(* CODESYS project PLC 1 Simulatie Structured Tekst 2V0 - Leeg.project
   Company: Avans
   Description: Simulatie voor opstelling Sorteer Station.
   Title: Simulatie Sorteer Station
   Author: Rene Potters/Gerard Harkema
   Version: 0.1.0

Project tree, tasks and I/O mapping:
  Device : CODESYS Control Win V3, 3S - Smart Software Solutions GmbH, version 3.5.13.20
    application SorteerStationSimulatie
      libraries: Standard, * (System); Util, * (System); VisuDialogs, 3.5.12.0 (System)
      task MainTask (cyclic, interval t#20ms, priority 1) calls Main
      task Simulatie (cyclic, interval t#20ms, priority 1) calls MagazijnSim, OverzetterSim, SorterenSim
  Device_1 : EHV-CPU1025, Hitachi-IES, order no. EHV-CPU1025, version 3.5.4.11
      settings: IP Address = '192.168.1.31'
    application SorteerStationRealWorld
      libraries: Standard, * (System); Util, * (System); VisuDialogs, 3.5.12.0 (System)
      task MainTask (cyclic, interval t#20ms, priority 1) calls Main
    Basic : Basic, Hitachi-IES, version 3.4.4.0
      <Empty>
      <Empty>
      <Empty>
      <Empty>
      <Empty>
      <Empty>
      <Empty>
      <Empty>
      <Empty>
      <Empty>
      <Empty>
  Simulatie/
    program MagazijnSim [ST]
    program SorterenSim [ST]
    global variables SIM
    program OverzetterSim [ST]
    data type OverzetterDUT
    data type SorterenDUT
    data type MagazijnDUT
    function block SorterenGootSim [ST]
  text list GlobalTextList
  Programma Structured Text/
    program Main [ST]
  global variables GVL
  Visualisaties/
    visualisation SorteerStationHMI
    visualisation BekerMagazijnHMI
    visualisation OverzetterHMI
    visualisation SorterenHMI
*)

// Simulatie/OverzetterDUT
{attribute 'qualified_only'}
{attribute 'strict'}
TYPE OverzetterDUT :
(
	INHETMIDDEN, NAARRECHTS, ISRECHTS, NAARLINKS, ISLINKS, GEVALLEN
);
END_TYPE

// Simulatie/SorterenDUT
{attribute 'qualified_only'}
{attribute 'strict'}
TYPE SorterenDUT :
(
	VOLGENDEBLOK, OPDEBAND, VOORSTOPPER, NAARGOOT1, INGOOT1, NAARGOOT2, INGOOT2, NAARGOOT3, INGOOT3, GEREED, VOL
);
END_TYPE

// Simulatie/MagazijnDUT
{attribute 'qualified_only'}
{attribute 'strict'}
TYPE MagazijnDUT :
(
	INGETROKKEN, INTREKKEN, UITGESTOTEN, UITSTOTEN, LEEG
);
END_TYPE

// Simulatie/SIM
{attribute 'qualified_only'}
VAR_GLOBAL
	// Rotatie van de overzetter
	Vx_OvzRotate: INT := 0;
	// Visualisatie invisible blok
	Vx_OvzBlokLinks: BOOL := FALSE;
	// Visualisatie invisible blok
	Vx_OvzBlokOverzetter: BOOL := FALSE;
	// Visualisatie invisible blok
	Vx_OvzBlokRechts: BOOL := FALSE;
	// Visualisatie invisible blok
	Vx_OvzBlokGevallen: BOOL := FALSE;	
	// Magazijn opnieuw vullen (simulatie)
	Ix_MagazijnVullen 	: BOOL;
	// Goten legen (symulatie)
	Ix_GotenLegen	  	: BOOL;
	
	
	
	
	
	
	
	
	
	
	
	
	
	
	
	
	
	
	
	
	
	
	
	
	
	
	
	
	
	
	
	
	
	
	
	
	
	
	
	
	
	
	
	
	
	
	
	
	// Simulatie visualisatie 
	Vw_Rotate45: INT := 45;
	// Visualisatie X positie van de uitstoter
	Vw_MagUitstoterBekerX: INT := 30;
	// Visualisatie invisible blok uitgestoten
	Vx_MagBlokUit: BOOL := TRUE;
	// Visualisatie invisible blok 1
	Vx_MagBlok1: BOOL := TRUE;
	// Visualisatie invisible blok 2
	Vx_MagBlok2: BOOL := TRUE;
	// Visualisatie invisible blok 3
	Vx_MagBlok3: BOOL := TRUE;
	// Visualisatie invisible blok 4
	Vx_MagBlok4: BOOL := TRUE;
	// Visualisatie invisible blokken
	Vx_MagBlok: ARRAY[1..8] OF BOOL;
	// Aantal blokken in het magazijn
	Vw_MagBlokAantal: INT := 4;
	// Simulatie onthoudt dat een blok maar 1x wordt uitgestoten
	Vw_MagBlok1X: INT := 0;
	// Ligt er een blok op band
	Vw_SorBlokBand: BOOL := FALSE;
	// Rotatie van de stopper
	Vw_SorStopperRotate: INT := 0;
	// Rotatie van de stopper goot 1
	Vw_SorGoot1Rotate: INT := 0;
	// Rotatie van de stopper goot 2
	Vw_SorGoot2Rotate: INT := 0;
	// Kleur van de blok op betreffende positie
	Vw_SorKleurBand: DWORD := 0;
	// Bewegen van de blok over de band
	Vi_SorBlokBandX: INT := 0;
	// Bewegen van de blok over de band
	Vi_SorBlokBandY: INT := 0;
	// Simulatie error. Inverse logica.
	Vx_MagLuchtDrukError: BOOL := TRUE;
	// Simulatie error. Inverse logica.
	Vx_MagIsInError: BOOL := TRUE;
	// Simulatie error. Inverse logica.
	Vx_MagIsUitError: BOOL := TRUE;
	// Simulatie error. Inverse logica.
	Vx_OvzLuchtDrukError: BOOL := TRUE;
	// Simulatie error. Inverse logica.
	Vx_OvzIsLinksError: BOOL := TRUE;
	// Simulatie error. Inverse logica.
	Vx_OvzIsRechtsError: BOOL := TRUE;
	// Simulatie error. Inverse logica.
	Vx_OvzVacuumError: BOOL := TRUE;
	// Simulatie error. Inverse logica.
	Vx_SorMotorAfvoerError: BOOL := TRUE;
	// Simulatie error. Inverse logica.
	Vx_SorGoot1InError: BOOL := TRUE;
	// Simulatie error. Inverse logica.
	Vx_SorGoot1UitError: BOOL := TRUE;
	// Simulatie error. Inverse logica.
	Vx_SorInGootError: BOOL := TRUE;
	// Ligt er een blok op de betreffende positie
	Vx_SorBlokGoot: ARRAY [1..3,1..6] OF BOOL;
	// Kleur van de blok op betreffende positie
	Vw_SorKleurGoot: ARRAY [1..3,1..6] OF DWORD;
END_VAR

// GVL
VAR_GLOBAL
	// Indrukken resetknop 
	Ix_Resetknop: BOOL;
	// Keuzeknop staat op hand
	Ix_Hand: BOOL;
	// Keuzeknop staat op auto
	Ix_Auto: BOOL;
	// Indrukken noodstop
	Ix_Noodstop: BOOL;
	// Bekers magazijn zijn op
	Ix_MagazijnLeeg: BOOL;
	// Beker is uit dekselmagazijn gestoten
	Ix_UitstoterBekerIn: BOOL;
	// Uitstoter Beker haalt nieuwe beker op
	Ix_UitstoterBekerUit: BOOL;
	// Indrukken startknop
	Ix_Stopknop: BOOL := TRUE;
	// Indrukken stopknop
	Ix_Startknop: BOOL;	
	//Perslucht is aanwezig
	Ix_PersluchtAanwezig :BOOL;
	//Werkstuk door overzetter opgepakt
	Ix_VacuumAanwezig :BOOL;
	//Overzetter haalt beker op(linker pos.)
	Ix_OverzetterIsLinks :BOOL;
	//Overzetter plaatst beker op sorteerpositie
	Ix_OverzetterIsRechts :BOOL;
	//Beker aanwezig op detectiepositie
	Ix_BekerAanwezig :BOOL;
	//Beker is van aluminium
	Ix_BekerMetaal :BOOL;
	//Beker reflecteert en is dus niet zwart
	Ix_BekerReflecteerd :BOOL;
	//Product is naar een van de goten gegaan
	Ix_BekerInGoot :BOOL;
	//Pusher uitvoergoot 1 is in
	Ix_UitvoerGoot1IsIn :BOOL;
	//Pusher uitvoergoot 2 is in
	Ix_UitvoerGoot2IsIn :BOOL;
	//Beker afvoeren is bezig
	Ix_StationAfvoerVrij :BOOL;
	//Pusher uitvoergoot 1 is uit
	Ix_UitvoerGoot1IsUit :BOOL;
	//Pusher uitvoergoot 2 is uit
	Ix_UitvoerGoot2IsUit :BOOL;
	// Beker uit magazijn stoten
	Qx_BekerUitstoten: BOOL;	
	//Beker oppakken
	Qx_VacuumAan :BOOL;
	//Beker loslaten
	Qx_BekerLossen :BOOL;
	//Overzetter naar bekermagazijn
	Qx_OverzetterLinks :BOOL;
	//Overzetter naar sorteerpositie
	Qx_OverzetterRechts :BOOL;
	//Transportband aan
	Qx_MotorAfvoerAan :BOOL;
	//Pusher goot 1 uit
	Qx_UitvoerGoot1Uit :BOOL;
	//Pusher goot 2 uit
	Qx_UitvoerGoot2Uit :BOOL;
	//Beker stoppen op band voor detectie
	Qx_StopperUit :BOOL;
	//Uitsorteren is bezet
	Qx_StationBezet :BOOL;
	// Visualisatie invisible Gele vlak
	Qx_GeleLamp: BOOL;
	// Visualisatie invisible groene vlak
	Qx_GroeneLamp: BOOL;
	// Visualisatie invisible rode vlak
	Qx_RodeLamp: BOOL;
END_VAR

// Programma Structured Text/Main
PROGRAM Main
VAR
END_VAR

END_PROGRAM

// Simulatie/MagazijnSim
PROGRAM MagazijnSim
VAR
	// Timer om uitstoten en intrekken te vertragen
	Fb_Pulse: BLINK;
	// Timer om intrekken te vertragen
	Fb_Trigger: F_TRIG;
	// Eerste keer om visualisatie te updaten
	Mx_FirstTime: BOOL := TRUE;
	// Afhandeling van het magazijn
	Me_MagState: MAGAZIJNDUT := MAGAZIJNDUT.INGETROKKEN;
END_VAR

//
// Common stuff.
//

IF (Mx_FirstTime) THEN
	SIM.Vw_MagBlokAantal := 8;
	SIM.Vx_MagBlokUit:= FALSE;
	
	Mx_FirstTime := FALSE;
END_IF

					
//
// Handle all pulse and trigger events.
//
Fb_Pulse(ENABLE:=TRUE,TIMELOW:=T#200MS, TIMEHIGH:=T#200MS);
Fb_Trigger(CLK:=Fb_Pulse.OUT);


//
// Only if no emergency active, start handling the simulation.
//
IF (SIM.Ix_MagazijnVullen) THEN
	Mx_FirstTime := TRUE;
	SIM.Ix_MagazijnVullen := FALSE;
	RETURN;
END_IF
	
//
// The pulse determines the speed of the cilinder to move in
// ore move out. The cilinder is only moved if the airpressure 
// is available.
//
IF (Fb_Trigger.Q AND SIM.Vx_MagLuchtDrukError) THEN
		
			
	CASE Me_MagState OF
		MAGAZIJNDUT.INGETROKKEN:
			IF (SIM.Vx_MagBlokUit) THEN
				SIM.Vw_MagBlokAantal := SIM.Vw_MagBlokAantal - 1;
			END_IF
		
			SIM.Vw_MagUitstoterBekerX := 1;
			SIM.Vw_MagBlok1X    	  := SIM.Vw_MagUitstoterBekerX;
			SIM.Vx_MagBlokUit         := FALSE;
	
			IF (Qx_BekerUitstoten) THEN
				Me_MagState := MAGAZIJNDUT.UITSTOTEN;
			END_IF

		MAGAZIJNDUT.INTREKKEN:
			SIM.Vw_MagUitstoterBekerX := SIM.Vw_MagUitstoterBekerX - 30;
			
			IF (SIM.Vw_MagUitstoterBekerX < 0) THEN 
				SIM.Vw_MagUitstoterBekerX := 0; 
			END_IF		
			
			IF (SIM.Vw_MagUitstoterBekerX = 0) THEN
				Me_MagState := MAGAZIJNDUT.INGETROKKEN;				
			END_IF		

			IF (Qx_BekerUitstoten) THEN
				Me_MagState := MAGAZIJNDUT.UITSTOTEN;
			END_IF	
	
		MAGAZIJNDUT.UITGESTOTEN:
			SIM.Vx_MagBlokUit         := SIM.Vx_MagBlok1;
						
			IF (NOT Qx_BekerUitstoten) THEN
				Me_MagState := MAGAZIJNDUT.INTREKKEN;
			END_IF	
		
		MAGAZIJNDUT.UITSTOTEN:
			SIM.Vw_MagUitstoterBekerX := SIM.Vw_MagUitstoterBekerX + 30;
			SIM.Vw_MagBlok1X    	  := SIM.Vw_MagUitstoterBekerX;			
		
			IF (SIM.Vw_MagUitstoterBekerX > 70) THEN
				Me_MagState := MAGAZIJNDUT.UITGESTOTEN;				
			END_IF		

			IF (NOT Qx_BekerUitstoten) THEN
				Me_MagState := MAGAZIJNDUT.INTREKKEN;
			END_IF	
		
	END_CASE

	GVL.Ix_UitstoterBekerIn  := (Me_MagState = MAGAZIJNDUT.INGETROKKEN) AND SIM.Vx_MagIsInError;
	GVL.Ix_UitstoterBekerUit := (Me_MagState = MAGAZIJNDUT.UITGESTOTEN) AND SIM.Vx_MagIsUitError;	
	GVL.Ix_MagazijnLeeg 	 := (SIM.Vw_MagBlokAantal <= 0) AND (Ix_UitstoterBekerIn);	
	
	SIM.Vx_MagBlok[8] := (SIM.Vw_MagBlokAantal >= 8);
	SIM.Vx_MagBlok[7] := (SIM.Vw_MagBlokAantal >= 7);
	SIM.Vx_MagBlok[6] := (SIM.Vw_MagBlokAantal >= 6);
	SIM.Vx_MagBlok[5] := (SIM.Vw_MagBlokAantal >= 5);		
	SIM.Vx_MagBlok[4] := (SIM.Vw_MagBlokAantal >= 4);
	SIM.Vx_MagBlok[3] := (SIM.Vw_MagBlokAantal >= 3);
	SIM.Vx_MagBlok[2] := (SIM.Vw_MagBlokAantal >= 2);
	SIM.Vx_MagBlok[1] := (SIM.Vw_MagBlokAantal >= 1);	
	
END_IF

END_PROGRAM

// Simulatie/OverzetterSim
PROGRAM OverzetterSim
VAR
	// Timer om overzetten te vertragen
	Fb_Pulse: BLINK;
	// Timer om overzetten te vertragen
	Fb_Trigger: F_TRIG;
	// Eerste keer om visualisatie te updaten
	Mx_FirstTime: BOOL := TRUE;
	// Afhandeling van de overzetter
	Me_OvzState: OverzetterDUT := OVERZETTERDUT.INHETMIDDEN;	
	// Afhandeling van het blokje
	Me_BlokState: OverzetterDUT := OVERZETTERDUT.INHETMIDDEN;	
	// Duurt even voor het vacuum aanwezig is
	Mi_VacuumCntr: INT := 0;	
END_VAR
VAR CONSTANT


	// Inverse logica
	INVISABLE: BOOL := TRUE;
	// Inverse logica
	VISABLE: BOOL := FALSE;

END_VAR

// Initialisatie.

IF (Mx_FirstTime) THEN
	Me_OvzState := OVERZETTERDUT.INHETMIDDEN;
	Me_BlokState := OVERZETTERDUT.ISLINKS;
	
	Mi_VacuumCntr := 0;
	SIM.Vx_OvzRotate := 0;
	Mx_FirstTime := FALSE;
END_IF

//
// Afhandelen van de pulse events. Hierdoor loopt de simulatie los van de 
// TASK tijd.
//
Fb_Pulse(ENABLE:=TRUE,TIMELOW:=T#100MS, TIMEHIGH:=T#100MS);
Fb_Trigger(CLK:=Fb_Pulse.OUT);


//
// Only if no emergency active, start handling the simulation.
//
IF (GVL.Ix_Noodstop) THEN
	Mx_FirstTime := TRUE;	
	RETURN;
END_IF
	
//
// The pulse determines the speed of the cilinder to move in
// ore move out. The cilinder is only moved if the airpressure 
// is available.
//
IF (Fb_Trigger.Q AND SIM.Vx_OvzLuchtDrukError) THEN
	
	//
	// De status van de arm wordt los afgehandeld van het blokje. De beweging
	// van de arm staat hier namelijk helemaal los van.
	//
	
	CASE Me_OvzState OF
		
		OVERZETTERDUT.INHETMIDDEN:
			// 
			// De arm is in beweging naar links of naar rechts.
			// Indien de arm in de uiterste positie is wordt er van 
			// state gewisseld. Aangezien de arm in beweging is staan
			// de eindschakelaars uit.
			//
			
			IF (GVL.Qx_OverzetterLinks) THEN
				IF (SIM.Vx_OvzRotate > -90) THEN
					GVL.Ix_OverzetterIsLinks := FALSE;	
					GVL.Ix_OverzetterIsRechts := FALSE;			
					SIM.Vx_OvzRotate := SIM.Vx_OvzRotate - 10;
				ELSE
					Me_OvzState := OVERZETTERDUT.ISLINKS;			
				END_IF	
				
			END_IF
				 
			IF (GVL.Qx_OverzetterRechts) THEN
				IF (SIM.Vx_OvzRotate < 90) THEN
					GVL.Ix_OverzetterIsLinks := FALSE;	
					GVL.Ix_OverzetterIsRechts := FALSE;				
					SIM.Vx_OvzRotate := SIM.Vx_OvzRotate + 10;
				ELSE
					Me_OvzState := OVERZETTERDUT.ISRECHTS;				
				END_IF			
			END_IF
				
		OVERZETTERDUT.ISLINKS:
		    //
			// Arm staat in een uiterste stand. Eindschakelaar is ingeschakeld.
			// Zodra de arm weer wordt bewogen verandert de state.
			//
			
			GVL.Ix_OverzetterIsLinks := TRUE AND SIM.Vx_OvzIsLinksError;	

			IF (GVL.Qx_OverzetterRechts AND NOT GVL.Qx_OverzetterLinks) THEN
				GVL.Ix_OverzetterIsLinks := FALSE;				
				Me_OvzState := OVERZETTERDUT.INHETMIDDEN;		
			END_IF
			
		OVERZETTERDUT.ISRECHTS:
		    //
			// Arm staat in een uiterste stand. Eindschakelaar is ingeschakeld.
			// Zodra de arm weer wordt bewogen verandert de state.
			//
		
			GVL.Ix_OverzetterIsRechts := TRUE AND SIM.Vx_OvzIsRechtsError;	

			IF (GVL.Qx_OverzetterLinks AND NOT GVL.Qx_OverzetterRechts) THEN
				GVL.Ix_OverzetterIsRechts := FALSE;				
				Me_OvzState := OVERZETTERDUT.INHETMIDDEN;		
			END_IF			
			
		END_CASE

	END_IF	

	//
	// De status van het blokje hangt af van een aantal stuursignalen zoals waar
	// de arm zich bevindt, of er vacuum is en of er een beker lossen wordt gegeven.
	//
	
	CASE Me_BlokState OF
		OVERZETTERDUT.ISLINKS:
			//
			// Als de arm links is moet er eerste een vacuum opgebouwd worden alvorens het blokje 
			// opgepakt kan worden. Daarna verandert de state. 
			//
			
			SIM.Vx_OvzBlokGevallen 	 := INVISABLE;
			SIM.Vx_OvzBlokLinks 	 := VISABLE;
			SIM.Vx_OvzBlokOverzetter := INVISABLE;
			SIM.Vx_OvzBlokRechts 	 := INVISABLE;
			
			IF (GVL.Qx_VacuumAan AND SIM.Vx_OvzVacuumError AND GVL.Ix_OverzetterIsLinks) AND (NOT GVL.Qx_BekerLossen) THEN
				Mi_VacuumCntr := Mi_VacuumCntr + 1;
			END_IF
			
			IF (NOT GVL.Qx_VacuumAan AND SIM.Vx_OvzVacuumError) THEN
				Mi_VacuumCntr := 0;
			END_IF

			GVL.Ix_VacuumAanwezig := (Mi_VacuumCntr > 50);
	
			IF  ( GVL.Ix_VacuumAanwezig AND (Me_OvzState = OVERZETTERDUT.INHETMIDDEN)) THEN
				Me_BlokState := OVERZETTERDUT.INHETMIDDEN;
			END_IF
			
		OVERZETTERDUT.INHETMIDDEN:
			//
			// Het blokje is in beweging zolang er vacuum is. Als er geen vacuum meer is
			// valt het blokje... Indien de arm helemaal rechts is kan het blokje gelost 
			// worden. Dit moet met een Bekerlossen ondanks het feit dat er
			// geen vacuum meer is....
			//
			
			SIM.Vx_OvzBlokGevallen 	 := INVISABLE;
			SIM.Vx_OvzBlokLinks 	 := INVISABLE;
			SIM.Vx_OvzBlokOverzetter := VISABLE;
			SIM.Vx_OvzBlokRechts 	 := INVISABLE;

		 	IF (GVL.Ix_OverzetterIsRechts) AND (NOT GVL.Qx_VacuumAan) AND (GVL.Qx_BekerLossen) THEN
				GVL.Ix_VacuumAanwezig := FALSE;
				Me_BlokState := OVERZETTERDUT.ISRECHTS;		
				RETURN;		
			END_IF
			
			IF (NOT GVL.Ix_OverzetterIsRechts) AND (NOT GVL.Ix_OverzetterIsLinks) AND(NOT GVL.Qx_VacuumAan) THEN
				GVL.Ix_VacuumAanwezig := FALSE;
				Me_BlokState := OVERZETTERDUT.GEVALLEN;				
			END_IF

		OVERZETTERDUT.ISRECHTS:	
		    // 
			// Blokje is gelost. Nu is het wachten tot de overzetter terug naar links wordt gestuurd. Daarna verdwijnt
			// het blokje automatisch.
			//
			
			SIM.Vx_OvzBlokGevallen 	 := INVISABLE;
			SIM.Vx_OvzBlokLinks 	 := INVISABLE;
			SIM.Vx_OvzBlokOverzetter := INVISABLE;
			SIM.Vx_OvzBlokRechts 	 := VISABLE;
			
			IF (NOT GVL.Ix_OverzetterIsRechts) THEN
				Me_BlokState := OVERZETTERDUT.ISLINKS;					
			END_IF

		OVERZETTERDUT.GEVALLEN:
			//
			// Blokje is gevallen..... Situatie herstelt zich zodra de arm helemaal links staat.
			//
				
			SIM.Vx_OvzBlokGevallen 	 := VISABLE;
			SIM.Vx_OvzBlokLinks 	 := INVISABLE;
			SIM.Vx_OvzBlokOverzetter := INVISABLE;
			SIM.Vx_OvzBlokRechts 	 := INVISABLE;
			
			IF (GVL.Ix_OverzetterIsLinks) THEN
				Me_BlokState := OVERZETTERDUT.ISLINKS;					
			END_IF				
	END_CASE

END_PROGRAM

// Simulatie/SorterenSim
PROGRAM SorterenSim
VAR
	// Timer om sorteren te vertragen
	Fb_Pulse: BLINK;
	// Timer om sorteren te vertragen
	Fb_Trigger: F_TRIG;
	// Eerste keer om visualisatie te updaten
	Mx_FirstTime: BOOL := TRUE;
	// Afhandeling van de overzetter
	Me_SorState: SORTERENDUT := SORTERENDUT.OPDEBAND;
	// Index voor posities
	Mi_PositieIndx: INT := 1;
	// Index voor goten.
	Mi_GootIndx: INT := 1;
	// Afhandeling blokjes in goot1.
	Mb_Goot1: SorterenGootSim;
	// Afhandeling blokjes in goot2.
	Mb_Goot2: SorterenGootSim;
	// Afhandeling blokjes in goot3.
	Mb_Goot3: SorterenGootSim;
	Mx_Geplaatst: BOOL := FALSE;
	// Random nummer om kleur te bepalen
	Mi_Random: UDINT := 1;	
END_VAR
VAR CONSTANT
	// Inverse logica
	INVISABLE: BOOL := TRUE;
	// Inverse logica
	VISABLE: BOOL := FALSE;
	// Kleur rood
	RED: DWORD := 16#00FF0000;
	// Kleur wit
	WHITE: DWORD := 16#00FFFFFF;
	// Stapgrootte voor bewegingen
	STEP: INT := 4;
	// Kleur zwart
	BLACK: DWORD := 16#00000000;
	// Kleur geel
	YELLOW: DWORD := 16#00FFFF00;
	// Goot 1
	GOOT1: INT := 1;
	// Goot 2
	GOOT2: INT := 2;
	// Goot 3
	GOOT3: INT := 3;
END_VAR

// Initialisatie.

IF (Mx_FirstTime) THEN
	Me_SorState := SORTERENDUT.VOLGENDEBLOK;

	SIM.Vw_SorBlokBand  := VISABLE;
	SIM.Vw_SorKleurBand := YELLOW;
	SIM.Vi_SorBlokBandX := 0;
	SIM.Vi_SorBlokBandY := 0;
	
	FOR Mi_GootIndx := 1 TO 3 DO 
		FOR Mi_PositieIndx := 1 TO 3 DO
			SIM.Vx_SorBlokGoot[Mi_GootIndx, Mi_PositieIndx ]  := INVISABLE;
			SIM.Vw_SorKleurGoot[Mi_GootIndx, Mi_PositieIndx ] := WHITE;			
		END_FOR
	END_FOR
 
	Mx_FirstTime := FALSE;
END_IF

//
// Afhandelen van de pulse events. Hierdoor loopt de simulatie los van de 
// TASK tijd.
//
Fb_Pulse(ENABLE:=TRUE,TIMELOW:=T#50MS, TIMEHIGH:=T#50MS);
Fb_Trigger(CLK:=Fb_Pulse.OUT);


//
// Only if no emergency active, start handling the simulation.
//
IF (SIM.Ix_GotenLegen) THEN
	Mx_FirstTime := TRUE;
	SIM.Ix_GotenLegen := FALSE;
	RETURN;
END_IF


// The pulse determines the speed of the cilinder to move in
// ore move out. The cilinder is only moved if the airpressure 
// is available.
//
IF (Fb_Trigger.Q) THEN
	IF (GVL.Qx_StopperUit) THEN
		SIM.Vw_SorStopperRotate := 90;
	ELSE
		SIM.Vw_SorStopperRotate := 0;		
	END_IF
	
	IF (GVL.Qx_UitvoerGoot1Uit) THEN
		SIM.Vw_SorGoot1Rotate := 45;
	ELSE
		SIM.Vw_SorGoot1Rotate := 0;		
	END_IF	

	GVL.Ix_UitvoerGoot1IsUit := (SIM.Vw_SorGoot1Rotate > 0) AND (SIM.Vx_SorGoot1UitError);
    GVL.Ix_UitvoerGoot1IsIn  := (SIM.Vw_SorGoot1Rotate = 0) AND (SIM.Vx_SorGoot1InError);	
	
	IF (GVL.Qx_UitvoerGoot2Uit) THEN
		SIM.Vw_SorGoot2Rotate := 45;
	ELSE
		SIM.Vw_SorGoot2Rotate := 0;		
	END_IF	

	GVL.Ix_UitvoerGoot2IsUit := (SIM.Vw_SorGoot2Rotate > 0);
    GVL.Ix_UitvoerGoot2IsIn  := (SIM.Vw_SorGoot2Rotate = 0);	
	
	GVL.Ix_BekerInGoot := SIM.Vx_SorInGootError AND NOT ((SIM.Vx_SorBlokGoot[1,1] = VISABLE) OR (SIM.Vx_SorBlokGoot[2,1] = VISABLE) OR (SIM.Vx_SorBlokGoot[3,1] = VISABLE) OR ((SIM.Vi_SorBlokBandY > 30) AND (SIM.Vi_SorBlokBandY < 40)));


				
	CASE Me_SorState OF
		SORTERENDUT.VOLGENDEBLOK:
			//
			// Zet alles klaar voor een volgende blokje.
			//

			Mi_Random := DINT_TO_UDINT(TIME_TO_DINT(TIME()));
			Mi_Random := SHR((Mi_Random AND 16#000000F00), 8); 
   
			IF (Mi_Random < 5) THEN
				SIM.Vw_SorKleurBand := RED;
			ELSE IF (Mi_Random < 10) THEN
					SIM.Vw_SorKleurBand := BLACK;
				ELSE 
					SIM.Vw_SorKleurBand := YELLOW;
				END_IF
			END_IF
			
			SIM.Vw_SorBlokBand := VISABLE;
			SIM.Vi_SorBlokBandX := 0;
			SIM.Vi_SorBlokBandY := 0;
	
			Me_SorState := SORTERENDUT.OPDEBAND;
		
		SORTERENDUT.OPDEBAND:
		
			//
			// Blokje ligt op de band. Verplaats tot voor de stopper.
			//
			
			IF ((GVL.Qx_MotorAfvoerAan) AND (SIM.Vx_SorMotorAfvoerError)) THEN
				SIM.Vi_SorBlokBandX := SIM.Vi_SorBlokBandX + STEP;
			END_IF
			
			GVL.Ix_StationAfvoerVrij := (SIM.Vi_SorBlokBandX < 20);
			
			IF (SIM.Vi_SorBlokBandX > 50) THEN
				Me_SorState := SORTERENDUT.VOORSTOPPER;
			END_IF
			
		SORTERENDUT.VOORSTOPPER: 
		
			//
			// Indien de stopper uit is, dan stopt het blokje en worden
			// de kleur sensoren geactiveerd. Anders loopt het blokje gewoon door
			// naar goot 1.
			//
			
			IF ((NOT GVL.Qx_StopperUit) AND (GVL.Qx_MotorAfvoerAan) AND (SIM.Vx_SorMotorAfvoerError)) THEN
				SIM.Vi_SorBlokBandX := SIM.Vi_SorBlokBandX + STEP;	
			END_IF

			IF (GVL.Qx_StopperUit) THEN
				GVL.Ix_BekerAanwezig := TRUE;
				GVL.Ix_BekerMetaal       := (SIM.Vw_SorKleurBand = YELLOW);
				GVL.Ix_BekerReflecteerd  := (SIM.Vw_SorKleurBand = YELLOW) OR (SIM.Vw_SorKleurBand = RED);
			END_IF
			
			
			IF (SIM.Vi_SorBlokBandX > 60) THEN
				Me_SorState := SORTERENDUT.NAARGOOT1;
			END_IF		
		
		
		SORTERENDUT.NAARGOOT1:
			//
			// Voor goot 1 wordt bepaald of de stopper uit staat en het blokje dus in de goot
			// gaat. Anders loopt het blokje door naar goot 2.
			//

			GVL.Ix_BekerAanwezig := FALSE;
			
			IF ((GVL.Qx_MotorAfvoerAan) AND (SIM.Vx_SorMotorAfvoerError)) THEN
				SIM.Vi_SorBlokBandX := SIM.Vi_SorBlokBandX + STEP;
			END_IF
			
			IF ((SIM.Vi_SorBlokBandX > 130) AND (GVL.Qx_MotorAfvoerAan) AND (SIM.Vx_SorMotorAfvoerError) AND (GVL.Qx_UitvoerGoot1Uit)) THEN
				Me_SorState := SORTERENDUT.INGOOT1;
			END_IF		
	
			IF ((SIM.Vi_SorBlokBandX > 130) AND (GVL.Qx_MotorAfvoerAan) AND (SIM.Vx_SorMotorAfvoerError) AND (NOT GVL.Qx_UitvoerGoot1Uit)) THEN
				Me_SorState := SORTERENDUT.NAARGOOT2;
			END_IF	
	 
		SORTERENDUT.INGOOT1:
			//
			// Blokje valt in goot 1. Hier kunnen 3 blokjes liggen. Het  blokje van de band beweegt de goot 
			// in en aan de hand van welke blokjes er al liggen wordt het eerst volgende blokje bepaald.
			// Dit blokje wordt vervolgens getoond. Daarna is het sorteren gereed. Let op dat de goot vol
			// melding even wordt getriggered als het blokje door de sensor valt.
			//
			
			IF (SIM.Vi_SorBlokBandX < 170) THEN
				SIM.Vi_SorBlokBandX := SIM.Vi_SorBlokBandX + 2*STEP;
			END_IF
			
			SIM.Vi_SorBlokBandY := SIM.Vi_SorBlokBandY + STEP;

			
			Mb_Goot1(Px_YPos:=SIM.Vi_SorBlokBandY, Px_Goot:=GOOT1);
		
			IF (Mb_Goot1.Px_Geplaatst) THEN
				Me_SorState := SORTERENDUT.GEREED;
			END_IF
			
			IF (SIM.Vx_SorBlokGoot[GOOT1, 1] = VISABLE) THEN
				Me_SorState := SORTERENDUT.VOL;
			END_IF
			
		SORTERENDUT.NAARGOOT2: 
			//
			// Voor goot 2 wordt bepaald of de stopper uit staat en het blokje dus in de goot
			// gaat. Anders loopt het blokje door naar goot 3.
			//
		
			IF ((GVL.Qx_MotorAfvoerAan) AND (SIM.Vx_SorMotorAfvoerError)) THEN
				SIM.Vi_SorBlokBandX := SIM.Vi_SorBlokBandX + STEP;
			END_IF
			
			IF ((SIM.Vi_SorBlokBandX > 230) AND (GVL.Qx_MotorAfvoerAan) AND (SIM.Vx_SorMotorAfvoerError) AND (GVL.Qx_UitvoerGoot2Uit)) THEN
				Me_SorState := SORTERENDUT.INGOOT2;
			END_IF		
	
			IF ((SIM.Vi_SorBlokBandX > 230) AND (GVL.Qx_MotorAfvoerAan) AND (SIM.Vx_SorMotorAfvoerError) AND (NOT GVL.Qx_UitvoerGoot2Uit)) THEN
				Me_SorState := SORTERENDUT.NAARGOOT3;
			END_IF	
		
		SORTERENDUT.INGOOT2:
	
			//
			// Blokje valt in goot 2. Hier kunnen 3 blokjes liggen. Het  blokje van de band beweegt de goot 
			// in en aan de hand van welke blokjes er al liggen wordt het eerst volgende blokje bepaald.
			// Dit blokje wordt vervolgens getoond. Daarna is het sorteren gereed. Let op dat de goot vol
			// melding even wordt getriggered als het blokje door de sensor valt.
			//
			
			IF (SIM.Vi_SorBlokBandX < 270) THEN
				SIM.Vi_SorBlokBandX := SIM.Vi_SorBlokBandX + 2*STEP;
			END_IF
			
			SIM.Vi_SorBlokBandY := SIM.Vi_SorBlokBandY + STEP;
					
			Mb_Goot2(Px_YPos:=SIM.Vi_SorBlokBandY, Px_Goot:=GOOT2);
		
			IF (Mb_Goot2.Px_Geplaatst) THEN
				Me_SorState := SORTERENDUT.GEREED;
			END_IF

			IF (SIM.Vx_SorBlokGoot[GOOT2, 1] = VISABLE) THEN
				Me_SorState := SORTERENDUT.VOL;
			END_IF
		
		SORTERENDUT.NAARGOOT3: 
			//
			// Er valt niks meer te stoppen. Blokje loopt door naar goot 3.
			//
		
			IF ((GVL.Qx_MotorAfvoerAan) AND (SIM.Vx_SorMotorAfvoerError)) THEN
				SIM.Vi_SorBlokBandX := SIM.Vi_SorBlokBandX + STEP;
			END_IF
			
			IF ((SIM.Vi_SorBlokBandX > 330) AND (GVL.Qx_MotorAfvoerAan) AND (SIM.Vx_SorMotorAfvoerError)) THEN
				Me_SorState := SORTERENDUT.INGOOT3;
			END_IF		
		
		SORTERENDUT.INGOOT3:
	
			//
			// Blokje valt in goot 3. Hier kunnen 3 blokjes liggen. Het  blokje van de band beweegt de goot 
			// in en aan de hand van welke blokjes er al liggen wordt het eerst volgende blokje bepaald.
			// Dit blokje wordt vervolgens getoond. Daarna is het sorteren gereed. Let op dat de goot vol
			// melding even wordt getriggered als het blokje door de sensor valt.
			//
			
			IF (SIM.Vi_SorBlokBandX < 370) THEN
				SIM.Vi_SorBlokBandX := SIM.Vi_SorBlokBandX + 2*STEP;
			END_IF
			
			SIM.Vi_SorBlokBandY := SIM.Vi_SorBlokBandY + STEP;
			
			Mb_Goot3(Px_YPos:=SIM.Vi_SorBlokBandY, Px_Goot:=GOOT3);
		
			IF (Mb_Goot3.Px_Geplaatst) THEN
				Me_SorState := SORTERENDUT.GEREED;
			END_IF
	
			IF (SIM.Vx_SorBlokGoot[GOOT3, 1] = VISABLE) THEN
				Me_SorState := SORTERENDUT.VOL;
			END_IF
		
		SORTERENDUT.GEREED:
			SIM.Vw_SorKleurBand := WHITE;
			SIM.Vw_SorBlokBand := INVISABLE;
			SIM.Vi_SorBlokBandX := 0;
			SIM.Vi_SorBlokBandY := 0;
			
			IF (NOT GVL.Qx_MotorAfvoerAan) THEN
				Me_SorState := SORTERENDUT.VOLGENDEBLOK;
			END_IF
			
		SORTERENDUT.VOL:
			RETURN;
			
	END_CASE

END_IF

END_PROGRAM

// Simulatie/SorterenGootSim
FUNCTION_BLOCK SorterenGootSim

VAR_INPUT
	// Huidige Y positie van de blok
	Px_YPos: INT;
	// Huidge goot
	Px_Goot: INT;
END_VAR
VAR
	// Index voor posities
	Mi_PositieIndx: INT := 1;	
	// Posities van de blokjes in de goot
	Mi_Posities: ARRAY[1..6] OF INT;	
END_VAR
VAR_OUTPUT
	// Er is een positie waar het blokje terecht komt.
	Px_Geplaatst: BOOL;
END_VAR
VAR
	// Eerste keer om visualisatie te updaten
	Mx_FirstTime: BOOL := TRUE;
END_VAR
VAR CONSTANT
	// Inverse logica
	INVISABLE: BOOL := TRUE;
	// Inverse logica
	VISABLE: BOOL := FALSE;

END_VAR


//
// Initialiseer de posities van de blokjes in de goot.
//

IF (Mx_FirstTime) THEN
	Mi_Posities[1] :=  40;
	Mi_Posities[2] :=  80;
	Mi_Posities[3] := 120;
	Mi_Posities[4] := 160;
	Mi_Posities[5] := 200;
	Mi_Posities[6] := 240;	
	
	Mx_FirstTime := FALSE;
END_IF

Px_Geplaatst := FALSE;

//
// Bepaal of de huidige positie van het blokje op de band dat in de goot valt
// past bij een vaste positie in de goot. Indien dit het geval is, neem dan 
// de kleur over en toon het blokje. De goot vult zich van onder naar boven.
//

FOR Mi_PositieIndx := 3 TO 1 BY -1 DO
	IF (SIM.Vx_SorBlokGoot[Px_Goot, Mi_PositieIndx] = INVISABLE) THEN
		IF (SIM.Vi_SorBlokBandY > Mi_Posities[Mi_PositieIndx] ) THEN
			SIM.Vx_SorBlokGoot[Px_Goot, Mi_PositieIndx]  := VISABLE;
			SIM.Vw_SorKleurGoot[Px_Goot, Mi_PositieIndx] := SIM.Vw_SorKleurBand;
			
			Px_Geplaatst := TRUE;
			RETURN;
		ELSE
			RETURN;
		END_IF
	END_IF
END_FOR

END_FUNCTION_BLOCK

// Visualisaties/SorteerStationHMI
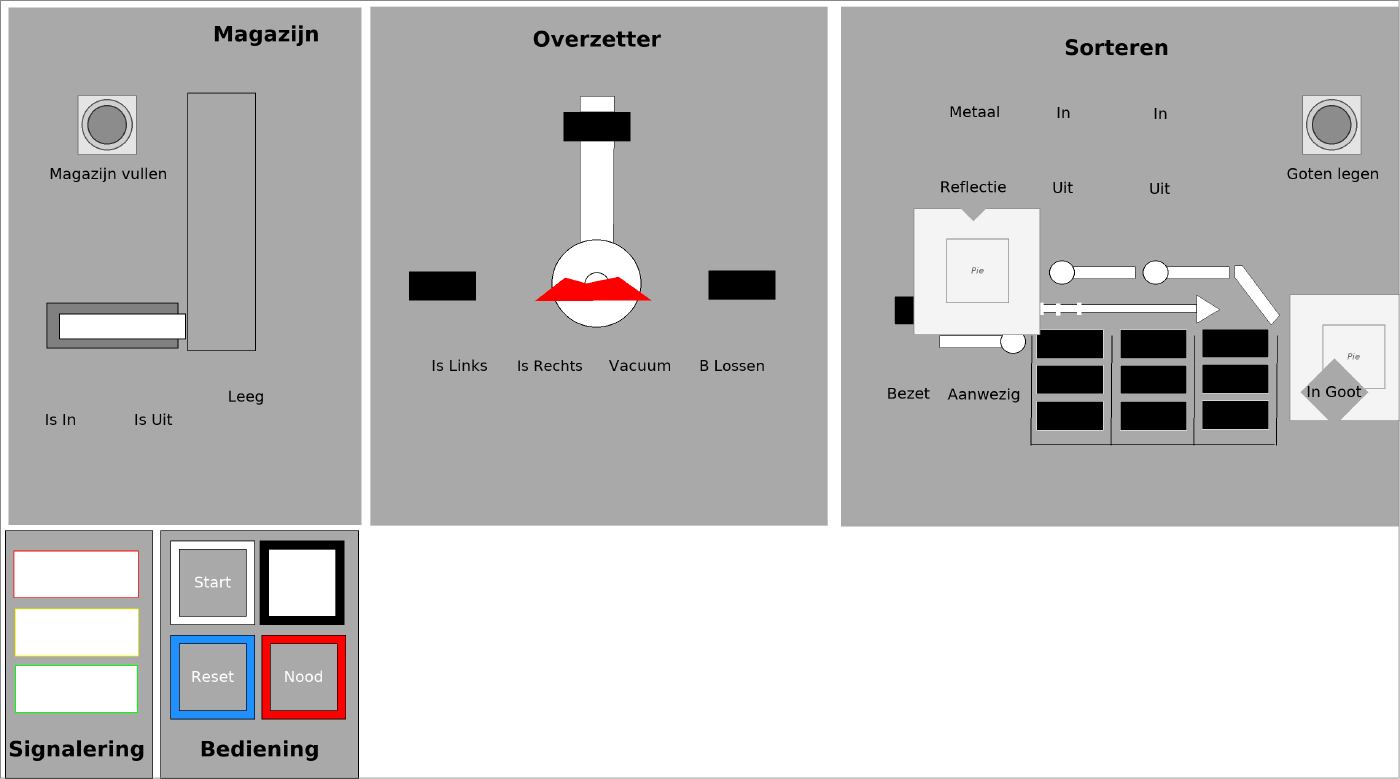
VISUALIZATION SorteerStationHMI  // 1660x924
    Rectangle (9,8 420x615)
    Polygon (247,458) (277,458) (307,458) (337,458) (292,538), "Leeg", colour toggle: Ix_MagazijnLeeg
    Polygon (72,458) (72,458) (112,498) (72,538) (32,498), "Is In", colour toggle: Ix_UitstoterBekerIn
    Polygon (182,458) (182,458) (222,498) (182,538) (142,498), "Is Uit", colour toggle: Ix_UitstoterBekerUit
    Rectangle (55,359 156x54)
    Rectangle (222,110 81x306)
    Rectangle (314,373 61x29), colour toggle: SIM.Vx_MagBlokUit
    Rectangle (227,338 61x29), colour toggle: SIM.Vx_MagBlok[2]
    Rectangle (227,302 61x29), colour toggle: SIM.Vx_MagBlok[3]
    Rectangle (227,266 61x29), colour toggle: SIM.Vx_MagBlok[4]
    Rectangle (227,373 61x29), colour toggle: SIM.Vx_MagBlok[1]
        p3560616238: SIM.Vw_MagBlok1X
    Rectangle (70,372 150x30)
        p3560616238: SIM.Vw_MagUitstoterBekerX
    Label (241,25 150x30), "Magazijn"
    Group (6,629 175x295)
        Rectangle (0,0 175x295)
        Rectangle (10,24 148x56), colour toggle: Qx_RodeLamp
        Rectangle (12,93 146x56), colour toggle: Qx_GeleLamp
        Rectangle (12,160 145x56), colour toggle: Qx_GroeneLamp
        Label (10,236 150x46), "Signalering"
    Group (190,629 235x295)
        Rectangle (0,0 235x295)
        Group (12,12 100x100)
            RoundedRectangle (0,0 100x100)
            RoundedRectangle (10,10 80x80), "Start", tooltip "Start knop", colour toggle: Ix_Startknop
                OnMouseDown: execute { Ix_Startknop := TRUE; }
                OnMouseUp: execute { Ix_Startknop := FALSE; }
        Group (118,12 100x100)
            RoundedRectangle (0,0 100x100)
            RoundedRectangle (10,10 80x80), "Stop", tooltip "Stop knop", colour toggle: Ix_Stopknop
                OnMouseDown: execute { Ix_Stopknop := FALSE; }
                OnMouseUp: execute { Ix_Stopknop := TRUE; }
        Group (12,124 100x100)
            RoundedRectangle (0,0 100x100)
            RoundedRectangle (10,10 80x80), "Reset", tooltip "Reset knop", colour toggle: Ix_Resetknop
                OnMouseDown: execute { Ix_Resetknop := TRUE; }
                OnMouseUp: execute { Ix_Resetknop := FALSE; }
        Group (120,124 100x100)
            RoundedRectangle (0,0 100x100), "Nood"
            RoundedRectangle (10,10 80x80), "Nood", tooltip "Noodstop", colour toggle: Ix_Noodstop
                OnMouseDown: execute { Ix_Noodstop := NOT Ix_Noodstop; }
        Label (43,236 150x46), "Bediening"
    Group (6,629 175x295)
        Rectangle (0,0 175x295)
        Rectangle (10,24 148x56), colour toggle: Qx_RodeLamp
        Rectangle (12,93 146x56), colour toggle: Qx_GeleLamp
        Rectangle (12,160 145x56), colour toggle: Qx_GroeneLamp
        Label (10,236 150x46), "Signalering"
    Group (190,629 235x295)
        Rectangle (0,0 235x295)
        Group (12,12 100x100)
            RoundedRectangle (0,0 100x100)
            RoundedRectangle (10,10 80x80), "Start", tooltip "Start knop", colour toggle: Ix_Startknop
                OnMouseDown: execute { Ix_Startknop := TRUE; }
                OnMouseUp: execute { Ix_Startknop := FALSE; }
        Group (118,12 100x100)
            RoundedRectangle (0,0 100x100)
            RoundedRectangle (10,10 80x80), "Stop", tooltip "Stop knop", colour toggle: Ix_Stopknop
                OnMouseDown: execute { Ix_Stopknop := FALSE; }
                OnMouseUp: execute { Ix_Stopknop := TRUE; }
        Group (12,124 100x100)
            RoundedRectangle (0,0 100x100)
            RoundedRectangle (10,10 80x80), "Reset", tooltip "Reset knop", colour toggle: Ix_Resetknop
                OnMouseDown: execute { Ix_Resetknop := TRUE; }
                OnMouseUp: execute { Ix_Resetknop := FALSE; }
        Group (120,124 100x100)
            RoundedRectangle (0,0 100x100), "Nood"
            RoundedRectangle (10,10 80x80), "Nood", tooltip "Noodstop", colour toggle: Ix_Noodstop
                OnMouseDown: execute { Ix_Noodstop := NOT Ix_Noodstop; }
        Label (43,236 150x46), "Bediening"
    Group (6,629 175x295)
        Rectangle (0,0 175x295)
        Rectangle (10,24 148x56), colour toggle: Qx_RodeLamp
        Rectangle (12,93 146x56), colour toggle: Qx_GeleLamp
        Rectangle (12,160 145x56), colour toggle: Qx_GroeneLamp
        Label (10,236 150x46), "Signalering"
    Rectangle (6,629 175x295)
    Rectangle (16,653 148x56), colour toggle: Qx_RodeLamp
    Rectangle (18,722 146x56), colour toggle: Qx_GeleLamp
    Rectangle (18,789 145x56), colour toggle: Qx_GroeneLamp
    Label (16,865 150x46), "Signalering"
    Group (190,629 235x295)
        Rectangle (0,0 235x295)
        Group (12,12 100x100)
            RoundedRectangle (0,0 100x100)
            RoundedRectangle (10,10 80x80), "Start", tooltip "Start knop", colour toggle: Ix_Startknop
                OnMouseDown: execute { Ix_Startknop := TRUE; }
                OnMouseUp: execute { Ix_Startknop := FALSE; }
        Group (118,12 100x100)
            RoundedRectangle (0,0 100x100)
            RoundedRectangle (10,10 80x80), "Stop", tooltip "Stop knop", colour toggle: Ix_Stopknop
                OnMouseDown: execute { Ix_Stopknop := FALSE; }
                OnMouseUp: execute { Ix_Stopknop := TRUE; }
        Group (12,124 100x100)
            RoundedRectangle (0,0 100x100)
            RoundedRectangle (10,10 80x80), "Reset", tooltip "Reset knop", colour toggle: Ix_Resetknop
                OnMouseDown: execute { Ix_Resetknop := TRUE; }
                OnMouseUp: execute { Ix_Resetknop := FALSE; }
        Group (120,124 100x100)
            RoundedRectangle (0,0 100x100), "Nood"
            RoundedRectangle (10,10 80x80), "Nood", tooltip "Noodstop", colour toggle: Ix_Noodstop
                OnMouseDown: execute { Ix_Noodstop := NOT Ix_Noodstop; }
        Label (43,236 150x46), "Bediening"
    Rectangle (190,629 235x295)
    Group (202,641 100x100)
        RoundedRectangle (0,0 100x100)
        RoundedRectangle (10,10 80x80), "Start", tooltip "Start knop", colour toggle: Ix_Startknop
            OnMouseDown: execute { Ix_Startknop := TRUE; }
            OnMouseUp: execute { Ix_Startknop := FALSE; }
    RoundedRectangle (202,641 100x100)
    RoundedRectangle (212,651 80x80), "Start", tooltip "Start knop", colour toggle: Ix_Startknop
        OnMouseDown: execute { Ix_Startknop := TRUE; }
        OnMouseUp: execute { Ix_Startknop := FALSE; }
    Group (308,641 100x100)
        RoundedRectangle (0,0 100x100)
        RoundedRectangle (10,10 80x80), "Stop", tooltip "Stop knop", colour toggle: Ix_Stopknop
            OnMouseDown: execute { Ix_Stopknop := FALSE; }
            OnMouseUp: execute { Ix_Stopknop := TRUE; }
    RoundedRectangle (308,641 100x100)
    RoundedRectangle (318,651 80x80), "Stop", tooltip "Stop knop", colour toggle: Ix_Stopknop
        OnMouseDown: execute { Ix_Stopknop := FALSE; }
        OnMouseUp: execute { Ix_Stopknop := TRUE; }
    Group (202,753 100x100)
        RoundedRectangle (0,0 100x100)
        RoundedRectangle (10,10 80x80), "Reset", tooltip "Reset knop", colour toggle: Ix_Resetknop
            OnMouseDown: execute { Ix_Resetknop := TRUE; }
            OnMouseUp: execute { Ix_Resetknop := FALSE; }
    RoundedRectangle (202,753 100x100)
    RoundedRectangle (212,763 80x80), "Reset", tooltip "Reset knop", colour toggle: Ix_Resetknop
        OnMouseDown: execute { Ix_Resetknop := TRUE; }
        OnMouseUp: execute { Ix_Resetknop := FALSE; }
    Group (310,753 100x100)
        RoundedRectangle (0,0 100x100), "Nood"
        RoundedRectangle (10,10 80x80), "Nood", tooltip "Noodstop", colour toggle: Ix_Noodstop
            OnMouseDown: execute { Ix_Noodstop := NOT Ix_Noodstop; }
    RoundedRectangle (310,753 100x100), "Nood"
    RoundedRectangle (320,763 80x80), "Nood", tooltip "Noodstop", colour toggle: Ix_Noodstop
        OnMouseDown: execute { Ix_Noodstop := NOT Ix_Noodstop; }
    Label (233,865 150x46), "Bediening"
    Rectangle (227,194 61x29), colour toggle: SIM.Vx_MagBlok[6]
    Rectangle (227,158 61x29), colour toggle: SIM.Vx_MagBlok[7]
    Rectangle (227,122 61x29), colour toggle: SIM.Vx_MagBlok[8]
    Rectangle (227,229 61x29), colour toggle: SIM.Vx_MagBlok[5]
    Rectangle (438,7 544x617)
    Polygon (545,394) (545,394) (585,434) (545,474) (505,434), "Is Links", colour toggle: Ix_OverzetterisLinks
    Polygon (652,394) (652,394) (692,434) (652,474) (612,434), "Is Rechts", colour toggle: Ix_OverzetterIsRechts
    Polygon (759,394) (759,394) (799,434) (759,474) (719,434), "Vacuum", colour toggle: Ix_VacuumAanwezig
    Polygon (688,131) (703,131) (728,131) (727,310) (688,310)
        p2858320360: SIM.Vx_OvzRotate
    Polygon (868,394) (868,394) (908,434) (868,474) (828,434), "B Lossen", colour toggle: Qx_BekerLossen
    Polygon (688,114) (703,114) (728,114) (728,132) (688,132), colour toggle: Qx_VacuumAan
        p2858320360: SIM.Vx_OvzRotate
    Polygon (668,133) (683,133) (747,133) (747,167) (668,167), invisible if: SIM.Vx_OvzBlokOverzetter
        p2277200375: SIM.Vx_OvzRotate
    Polygon (485,322) (500,322) (564,322) (564,356) (485,356), invisible if: SIM.Vx_OvzBlokLinks
    Polygon (840,321) (855,321) (919,321) (919,355) (840,355), invisible if: SIM.Vx_OvzBlokRechts
    Ellipse (654,284 106x104)
    Ellipse (693,323 29x27)
    Polygon (670,329) (695,336) (733,328) (772,356) (634,357), invisible if: SIM.Vx_OvzBlokGevallen
        p2277200375: SIM.Vx_OvzRotate
    Label (606,31 204x30), "Overzetter"
    Rectangle (996,7 664x618)
    Group (1197,350 249x33)
        Rectangle (0,11 222x10), colour toggle: GVL.Qx_MotorAfvoerAan
        Polygon (222,9) (222,0) (249,17) (222,33) (222,22), colour toggle: GVL.Qx_MotorAfvoerAan
        Rectangle (4,9 5x14)
        Rectangle (18,9 5x14)
        Rectangle (35,9 5x14)
        Rectangle (55,10 5x14)
        Rectangle (80,9 5x14)
    Polygon (1261,94) (1261,94) (1301,134) (1261,174) (1221,134), "In", colour toggle: GVL.Ix_UitvoerGoot1IsIn
    Polygon (1260,183) (1260,183) (1300,223) (1260,263) (1220,223), "Uit", colour toggle: GVL.Ix_UitvoerGoot1IsUit
    Polygon (1060,351) (1075,351) (1139,351) (1139,385) (1060,385), invisible if: SIM.Vw_SorBlokBand, colour variable: SIM.Vw_SorKleurBand
        p3560616238: SIM.Vi_SorBlokBandX
        p2738717112: SIM.Vi_SorBlokBandY
    Polygon (1229,391) (1244,391) (1308,391) (1308,425) (1229,425), invisible if: SIM.Vx_SorBlokGoot[1,1], colour variable: SIM.Vw_SorKleurGoot[1,1]
    Polygon (1229,433) (1244,433) (1308,433) (1308,467) (1229,467), invisible if: SIM.Vx_SorBlokGoot[1,2], colour variable: SIM.Vw_SorKleurGoot[1,2]
    Polygon (1229,476) (1244,476) (1308,476) (1308,510) (1229,510), invisible if: SIM.Vx_SorBlokGoot[1,3], colour variable: SIM.Vw_SorKleurGoot[1,3]
    Polygon (1328,391) (1343,391) (1407,391) (1407,425) (1328,425), invisible if: SIM.Vx_SorBlokGoot[2,1], colour variable: SIM.Vw_SorKleurGoot[2,1]
    Polygon (1328,433) (1343,433) (1407,433) (1407,467) (1328,467), invisible if: SIM.Vx_SorBlokGoot[2,2], colour variable: SIM.Vw_SorKleurGoot[2,2]
    Polygon (1328,476) (1343,476) (1407,476) (1407,510) (1328,510), invisible if: SIM.Vx_SorBlokGoot[2,3], colour variable: SIM.Vw_SorKleurGoot[2,3]
    Polygon (1425,390) (1440,390) (1504,390) (1504,424) (1425,424), invisible if: SIM.Vx_SorBlokGoot[3,1], colour variable: SIM.Vw_SorKleurGoot[3,1]
    Polygon (1425,432) (1440,432) (1504,432) (1504,466) (1425,466), invisible if: SIM.Vx_SorBlokGoot[3,2], colour variable: SIM.Vw_SorKleurGoot[3,2]
    Polygon (1425,475) (1440,475) (1504,475) (1504,509) (1425,509), invisible if: SIM.Vx_SorBlokGoot[3,3], colour variable: SIM.Vw_SorKleurGoot[3,3]
    Polygon (1114,398) (1169,398) (1192,398) (1192,412) (1114,412)
        p2858320360: SIM.Vw_SorStopperRotate
    Ellipse (1186,391 30x28)
    Polygon (1268,316) (1323,316) (1346,316) (1346,330) (1268,330)
        p2858320360: SIM.Vw_SorGoot1Rotate
    Ellipse (1244,309 30x28)
    Polygon (1379,316) (1434,316) (1457,316) (1457,330) (1379,330)
        p2858320360: SIM.Vw_SorGoot2Rotate
    Ellipse (1355,309 30x28)
    Polygon (1464,315) (1473,315) (1517,374) (1507,385) (1464,329)
    Group (1083,247 80x82)
        Pie (0,0 150x150)
        Pie (39,36 74x76)
    Line (1223,398) (1222,528)
    Line (1318,398) (1317,528)
    Line (1416,398) (1415,528)
    Line (1514,398) (1513,528)
    Line (1223,527) (1511,527)
    Group (1529,349 65x105)
        Pie (0,0 150x150)
        Pie (39,36 74x76)
    Polygon (1376,95) (1376,95) (1416,135) (1376,175) (1336,135), "In", colour toggle: GVL.Ix_UitvoerGoot2IsIn
    Polygon (1375,184) (1375,184) (1415,224) (1375,264) (1335,224), "Uit", colour toggle: GVL.Ix_UitvoerGoot2IsUit
    Polygon (1582,425) (1582,425) (1622,465) (1582,505) (1542,465), "In Goot", colour toggle: GVL.Ix_BekerInGoot
    Polygon (1077,427) (1077,427) (1117,467) (1077,507) (1037,467), "Bezet", colour toggle: GVL.Ix_StationAfvoerVrij
    Polygon (1156,93) (1156,93) (1196,133) (1156,173) (1116,133), "Metaal", colour toggle: GVL.Ix_BekerMetaal
    Polygon (1154,182) (1154,182) (1194,222) (1154,262) (1114,222), "Reflectie", colour toggle: GVL.Ix_BekerReflecteerd
    Polygon (1172,428) (1172,428) (1212,468) (1172,508) (1122,468), "Aanwezig", colour toggle: GVL.Ix_BekerAanwezig
    Label (1249,41 150x30), "Sorteren"
    Polygon (51,194) (81,194) (111,194) (206,208) (106,222), "Magazijn vullen", colour toggle: Ix_MagazijnLeeg
    PushSwitch (92,113 70x70), tooltip "Magazijn vullen", variable: SIM.Ix_MagazijnVullen, behaviour: TOGGLE, style: Switch-PushSwitch-Gray
    Polygon (1503,194) (1533,194) (1563,194) (1658,208) (1558,222), "Goten legen", colour toggle: Ix_MagazijnLeeg
    PushSwitch (1544,113 70x70), tooltip "Goten legen", variable: SIM.Ix_GotenLegen, behaviour: TOGGLE, style: Switch-PushSwitch-Gray
END_VISUALIZATION

// Visualisaties/BekerMagazijnHMI
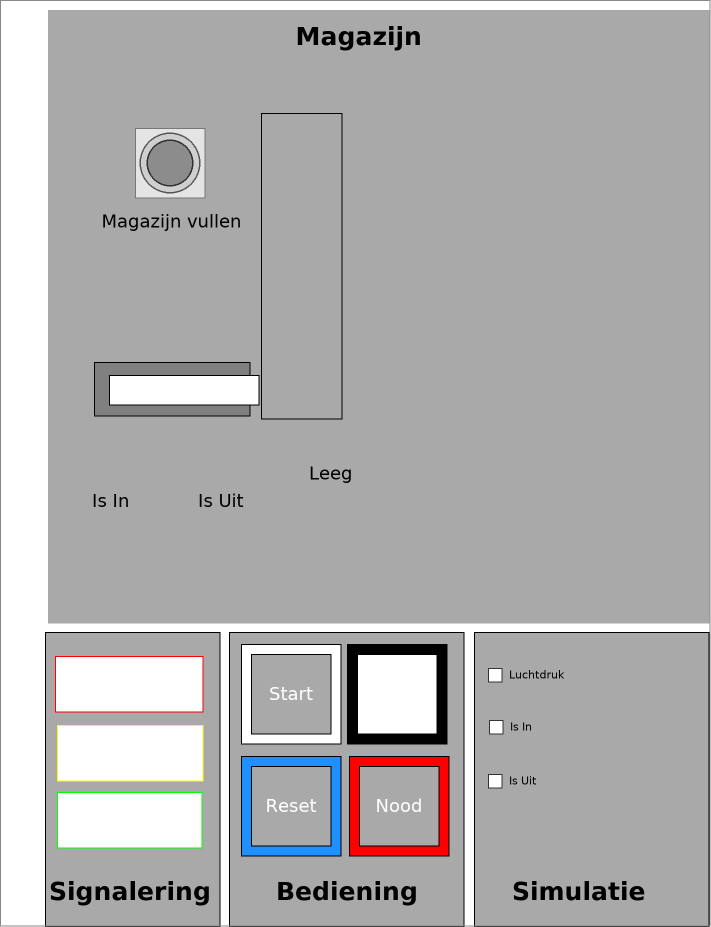
VISUALIZATION BekerMagazijnHMI  // 711x927
    Rectangle (47,9 664x615)
    Polygon (286,461) (316,461) (346,461) (376,461) (331,541), "Leeg", colour toggle: Ix_MagazijnLeeg
    Polygon (111,461) (111,461) (151,501) (111,541) (71,501), "Is In", colour toggle: Ix_UitstoterBekerIn
    Polygon (221,461) (221,461) (261,501) (221,541) (181,501), "Is Uit", colour toggle: Ix_UitstoterBekerUit
    Rectangle (94,362 156x54)
    Rectangle (261,113 81x306)
    Rectangle (353,376 61x29), colour toggle: SIM.Vx_MagBlokUit
    Rectangle (266,341 61x29), colour toggle: SIM.Vx_MagBlok[2]
    Rectangle (266,305 61x29), colour toggle: SIM.Vx_MagBlok[3]
    Rectangle (266,269 61x29), colour toggle: SIM.Vx_MagBlok[4]
    Rectangle (266,376 61x29), colour toggle: SIM.Vx_MagBlok[1]
        p3560616238: SIM.Vw_MagBlok1X
    Rectangle (109,375 150x30)
        p3560616238: SIM.Vw_MagUitstoterBekerX
    Label (284,21 150x30), "Magazijn"
    Group (45,632 664x295)
        Group (0,0 664x295)
            Group (429,0 235x295)
                Rectangle (0,0 235x295)
                Label (30,236 150x46), "Simulatie"
            Group (0,0 175x295)
                Rectangle (0,0 175x295)
                Rectangle (10,24 148x56), colour toggle: Qx_RodeLamp
                Rectangle (12,93 146x56), colour toggle: Qx_GeleLamp
                Rectangle (12,160 145x56), colour toggle: Qx_GroeneLamp
                Label (10,236 150x46), "Signalering"
            Group (184,0 235x295)
                Rectangle (0,0 235x295)
                Group (12,12 100x100)
                    RoundedRectangle (0,0 100x100)
                    RoundedRectangle (10,10 80x80), "Start", tooltip "Start knop", colour toggle: Ix_Startknop
                        OnMouseDown: execute { Ix_Startknop := TRUE; }
                        OnMouseUp: execute { Ix_Startknop := FALSE; }
                Group (118,12 100x100)
                    RoundedRectangle (0,0 100x100)
                    RoundedRectangle (10,10 80x80), "Stop", tooltip "Stop knop", colour toggle: Ix_Stopknop
                        OnMouseDown: execute { Ix_Stopknop := FALSE; }
                        OnMouseUp: execute { Ix_Stopknop := TRUE; }
                Group (12,124 100x100)
                    RoundedRectangle (0,0 100x100)
                    RoundedRectangle (10,10 80x80), "Reset", tooltip "Reset knop", colour toggle: Ix_Resetknop
                        OnMouseDown: execute { Ix_Resetknop := TRUE; }
                        OnMouseUp: execute { Ix_Resetknop := FALSE; }
                Group (120,124 100x100)
                    RoundedRectangle (0,0 100x100), "Nood"
                    RoundedRectangle (10,10 80x80), "Nood", tooltip "Noodstop", colour toggle: Ix_Noodstop
                        OnMouseDown: execute { Ix_Noodstop := NOT Ix_Noodstop; }
                Label (43,236 150x46), "Bediening"
        Checkbox (441,17 196x52), "Luchtdruk", variable: SIM.Vx_MagLuchtDrukError
        Checkbox (442,69 196x52), "Is In", variable: SIM.Vx_MagIsInError
        Checkbox (441,123 196x52), "Is Uit", variable: SIM.Vx_MagIsUitError
    Rectangle (266,197 61x29), colour toggle: SIM.Vx_MagBlok[6]
    Rectangle (266,161 61x29), colour toggle: SIM.Vx_MagBlok[7]
    Rectangle (266,125 61x29), colour toggle: SIM.Vx_MagBlok[8]
    Rectangle (266,232 61x29), colour toggle: SIM.Vx_MagBlok[5]
    PushSwitch (135,128 70x70), tooltip "Magazijn vullen", variable: SIM.Ix_MagazijnVullen, behaviour: TOGGLE, style: Switch-PushSwitch-Gray
    Polygon (94,209) (124,209) (154,209) (249,223) (149,237), "Magazijn vullen", colour toggle: Ix_MagazijnLeeg
END_VISUALIZATION

// Visualisaties/OverzetterHMI
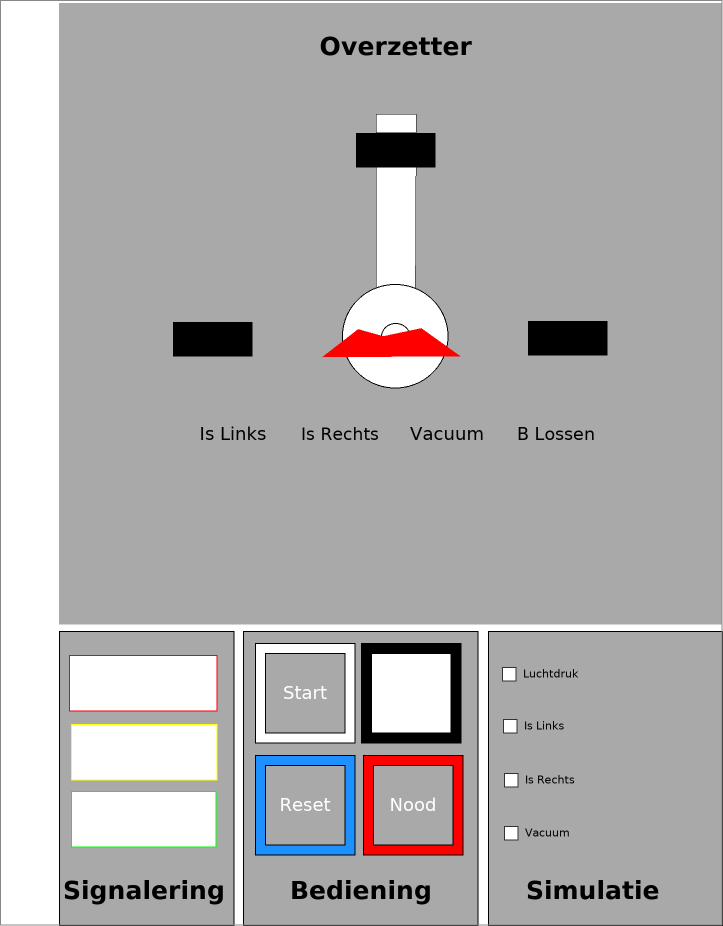
VISUALIZATION OverzetterHMI  // 723x926
    Rectangle (58,2 664x623)
    Polygon (233,394) (233,394) (273,434) (233,474) (193,434), "Is Links", colour toggle: Ix_OverzetterisLinks
    Polygon (340,394) (340,394) (380,434) (340,474) (300,434), "Is Rechts", colour toggle: Ix_OverzetterIsRechts
    Polygon (447,394) (447,394) (487,434) (447,474) (407,434), "Vacuum", colour toggle: Ix_VacuumAanwezig
    Polygon (376,131) (391,131) (416,131) (415,310) (376,310)
        p2858320360: SIM.Vx_OvzRotate
    Polygon (556,394) (556,394) (596,434) (556,474) (516,434), "B Lossen", colour toggle: Qx_BekerLossen
    Polygon (376,114) (391,114) (416,114) (416,132) (376,132), colour toggle: Qx_VacuumAan
        p2858320360: SIM.Vx_OvzRotate
    Polygon (356,133) (371,133) (435,133) (435,167) (356,167), invisible if: SIM.Vx_OvzBlokOverzetter
        p2277200375: SIM.Vx_OvzRotate
    Polygon (173,322) (188,322) (252,322) (252,356) (173,356), invisible if: SIM.Vx_OvzBlokLinks
    Polygon (528,321) (543,321) (607,321) (607,355) (528,355), invisible if: SIM.Vx_OvzBlokRechts
    Ellipse (342,284 106x104)
    Ellipse (381,323 29x27)
    Polygon (358,329) (383,336) (421,328) (460,356) (322,357), invisible if: SIM.Vx_OvzBlokGevallen
        p2277200375: SIM.Vx_OvzRotate
    Label (294,31 204x30), "Overzetter"
    Group (59,631 175x295)
        Rectangle (0,0 175x295)
        Rectangle (10,24 148x56), colour toggle: Qx_RodeLamp
        Rectangle (12,93 146x56), colour toggle: Qx_GeleLamp
        Rectangle (12,160 145x56), colour toggle: Qx_GroeneLamp
        Label (10,236 150x46), "Signalering"
    Group (243,631 235x295)
        Rectangle (0,0 235x295)
        Group (12,12 100x100)
            RoundedRectangle (0,0 100x100)
            RoundedRectangle (10,10 80x80), "Start", tooltip "Start knop", colour toggle: Ix_Startknop
                OnMouseDown: execute { Ix_Startknop := TRUE; }
                OnMouseUp: execute { Ix_Startknop := FALSE; }
        Group (118,12 100x100)
            RoundedRectangle (0,0 100x100)
            RoundedRectangle (10,10 80x80), "Stop", tooltip "Stop knop", colour toggle: Ix_Stopknop
                OnMouseDown: execute { Ix_Stopknop := FALSE; }
                OnMouseUp: execute { Ix_Stopknop := TRUE; }
        Group (12,124 100x100)
            RoundedRectangle (0,0 100x100)
            RoundedRectangle (10,10 80x80), "Reset", tooltip "Reset knop", colour toggle: Ix_Resetknop
                OnMouseDown: execute { Ix_Resetknop := TRUE; }
                OnMouseUp: execute { Ix_Resetknop := FALSE; }
        Group (120,124 100x100)
            RoundedRectangle (0,0 100x100), "Nood"
            RoundedRectangle (10,10 80x80), "Nood", tooltip "Noodstop", colour toggle: Ix_Noodstop
                OnMouseDown: execute { Ix_Noodstop := NOT Ix_Noodstop; }
        Label (43,236 150x46), "Bediening"
    Group (488,631 235x295)
        Group (0,0 235x295)
            Rectangle (0,0 235x295)
            Label (30,236 150x46), "Simulatie"
        Checkbox (12,17 196x52), "Luchtdruk", variable: SIM.Vx_OvzLuchtDrukError
        Checkbox (13,69 196x52), "Is Links", variable: SIM.Vx_OvzIsLinksError
        Checkbox (14,123 196x52), "Is Rechts", variable: SIM.Vx_OvzIsRechtsError
        Checkbox (14,176 196x52), "Vacuum", variable: SIM.Vx_OvzVacuumError
END_VISUALIZATION

// Visualisaties/SorterenHMI
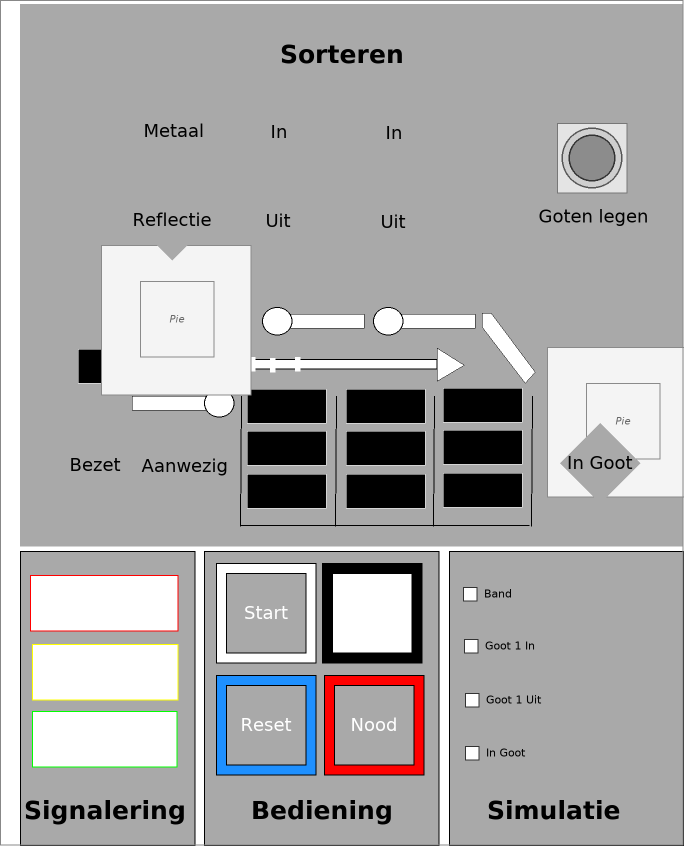
VISUALIZATION SorterenHMI  // 684x846
    Rectangle (19,3 664x544)
    Group (215,348 249x33)
        Rectangle (0,11 222x10), colour toggle: GVL.Qx_MotorAfvoerAan
        Polygon (222,9) (222,0) (249,17) (222,33) (222,22), colour toggle: GVL.Qx_MotorAfvoerAan
        Rectangle (4,9 5x14)
        Rectangle (18,9 5x14)
        Rectangle (35,9 5x14)
        Rectangle (55,10 5x14)
        Rectangle (80,9 5x14)
    Polygon (279,92) (279,92) (319,132) (279,172) (239,132), "In", colour toggle: GVL.Ix_UitvoerGoot1IsIn
    Polygon (278,181) (278,181) (318,221) (278,261) (238,221), "Uit", colour toggle: GVL.Ix_UitvoerGoot1IsUit
    Polygon (78,349) (93,349) (157,349) (157,383) (78,383), invisible if: SIM.Vw_SorBlokBand, colour variable: SIM.Vw_SorKleurBand
        p3560616238: SIM.Vi_SorBlokBandX
        p2738717112: SIM.Vi_SorBlokBandY
    Polygon (247,389) (262,389) (326,389) (326,423) (247,423), invisible if: SIM.Vx_SorBlokGoot[1,1], colour variable: SIM.Vw_SorKleurGoot[1,1]
    Polygon (247,431) (262,431) (326,431) (326,465) (247,465), invisible if: SIM.Vx_SorBlokGoot[1,2], colour variable: SIM.Vw_SorKleurGoot[1,2]
    Polygon (247,474) (262,474) (326,474) (326,508) (247,508), invisible if: SIM.Vx_SorBlokGoot[1,3], colour variable: SIM.Vw_SorKleurGoot[1,3]
    Polygon (346,389) (361,389) (425,389) (425,423) (346,423), invisible if: SIM.Vx_SorBlokGoot[2,1], colour variable: SIM.Vw_SorKleurGoot[2,1]
    Polygon (346,431) (361,431) (425,431) (425,465) (346,465), invisible if: SIM.Vx_SorBlokGoot[2,2], colour variable: SIM.Vw_SorKleurGoot[2,2]
    Polygon (346,474) (361,474) (425,474) (425,508) (346,508), invisible if: SIM.Vx_SorBlokGoot[2,3], colour variable: SIM.Vw_SorKleurGoot[2,3]
    Polygon (443,388) (458,388) (522,388) (522,422) (443,422), invisible if: SIM.Vx_SorBlokGoot[3,1], colour variable: SIM.Vw_SorKleurGoot[3,1]
    Polygon (443,430) (458,430) (522,430) (522,464) (443,464), invisible if: SIM.Vx_SorBlokGoot[3,2], colour variable: SIM.Vw_SorKleurGoot[3,2]
    Polygon (443,473) (458,473) (522,473) (522,507) (443,507), invisible if: SIM.Vx_SorBlokGoot[3,3], colour variable: SIM.Vw_SorKleurGoot[3,3]
    Polygon (132,396) (187,396) (210,396) (210,410) (132,410)
        p2858320360: SIM.Vw_SorStopperRotate
    Ellipse (204,389 30x28)
    Polygon (286,314) (341,314) (364,314) (364,328) (286,328)
        p2858320360: SIM.Vw_SorGoot1Rotate
    Ellipse (262,307 30x28)
    Polygon (397,314) (452,314) (475,314) (475,328) (397,328)
        p2858320360: SIM.Vw_SorGoot2Rotate
    Ellipse (373,307 30x28)
    Polygon (482,313) (491,313) (535,372) (525,383) (482,327)
    Group (101,245 80x82)
        Pie (0,0 150x150)
        Pie (39,36 74x76)
    Line (241,396) (240,526)
    Line (336,396) (335,526)
    Line (434,396) (433,526)
    Line (532,396) (531,526)
    Line (241,525) (529,525)
    Group (547,347 65x105)
        Pie (0,0 150x150)
        Pie (39,36 74x76)
    Polygon (394,93) (394,93) (434,133) (394,173) (354,133), "In", colour toggle: GVL.Ix_UitvoerGoot2IsIn
    Polygon (393,182) (393,182) (433,222) (393,262) (353,222), "Uit", colour toggle: GVL.Ix_UitvoerGoot2IsUit
    Polygon (600,423) (600,423) (640,463) (600,503) (560,463), "In Goot", colour toggle: GVL.Ix_BekerInGoot
    Polygon (95,425) (95,425) (135,465) (95,505) (55,465), "Bezet", colour toggle: GVL.Ix_StationAfvoerVrij
    Polygon (174,91) (174,91) (214,131) (174,171) (134,131), "Metaal", colour toggle: GVL.Ix_BekerMetaal
    Polygon (172,180) (172,180) (212,220) (172,260) (132,220), "Reflectie", colour toggle: GVL.Ix_BekerReflecteerd
    Polygon (190,426) (190,426) (230,466) (190,506) (140,466), "Aanwezig", colour toggle: GVL.Ix_BekerAanwezig
    Label (267,39 150x30), "Sorteren"
    Group (20,551 175x295)
        Rectangle (0,0 175x295)
        Rectangle (10,24 148x56), colour toggle: Qx_RodeLamp
        Rectangle (12,93 146x56), colour toggle: Qx_GeleLamp
        Rectangle (12,160 145x56), colour toggle: Qx_GroeneLamp
        Label (10,236 150x46), "Signalering"
    Group (204,551 235x295)
        Rectangle (0,0 235x295)
        Group (12,12 100x100)
            RoundedRectangle (0,0 100x100)
            RoundedRectangle (10,10 80x80), "Start", tooltip "Start knop", colour toggle: Ix_Startknop
                OnMouseDown: execute { Ix_Startknop := TRUE; }
                OnMouseUp: execute { Ix_Startknop := FALSE; }
        Group (118,12 100x100)
            RoundedRectangle (0,0 100x100)
            RoundedRectangle (10,10 80x80), "Stop", tooltip "Stop knop", colour toggle: Ix_Stopknop
                OnMouseDown: execute { Ix_Stopknop := FALSE; }
                OnMouseUp: execute { Ix_Stopknop := TRUE; }
        Group (12,124 100x100)
            RoundedRectangle (0,0 100x100)
            RoundedRectangle (10,10 80x80), "Reset", tooltip "Reset knop", colour toggle: Ix_Resetknop
                OnMouseDown: execute { Ix_Resetknop := TRUE; }
                OnMouseUp: execute { Ix_Resetknop := FALSE; }
        Group (120,124 100x100)
            RoundedRectangle (0,0 100x100), "Nood"
            RoundedRectangle (10,10 80x80), "Nood", tooltip "Noodstop", colour toggle: Ix_Noodstop
                OnMouseDown: execute { Ix_Noodstop := NOT Ix_Noodstop; }
        Label (43,236 150x46), "Bediening"
    Group (449,551 235x295)
        Group (0,0 235x295)
            Rectangle (0,0 235x295)
            Label (30,236 150x46), "Simulatie"
        Checkbox (12,17 196x52), "Band", variable: SIM.Vx_SorMotorAfvoerError
        Checkbox (13,69 196x52), "Goot 1 In", variable: SIM.Vx_SorGoot1InError
        Checkbox (14,123 196x52), "Goot 1 Uit", variable: SIM.Vx_SorGoot1UitError
        Checkbox (14,176 196x52), "In Goot", variable: SIM.Vx_SorGoot1InError
    PushSwitch (557,123 70x70), tooltip "Goten legen", variable: SIM.Ix_GotenLegen, behaviour: TOGGLE, style: Switch-PushSwitch-Gray
    Polygon (516,204) (546,204) (576,204) (671,218) (571,232), "Goten legen", colour toggle: Ix_MagazijnLeeg
END_VISUALIZATION
